Fanuc TP program (LS listing): stripped_lines.ls

/PROG  STRIPPED_TEST
/ATTR
OWNER		= MNEDITOR;
COMMENT		= "";
PROG_SIZE	= 548;
CREATE		= DATE 24-01-23  TIME 05:57:44;
MODIFIED	= DATE 25-09-11  TIME 00:54:24;
FILE_NAME	= ;
VERSION		= 0;
LINE_COUNT	= 5;
MEMORY_SIZE	= 940;
PROTECT		= READ_WRITE;
TCD:  STACK_SIZE	= 0,
      TASK_PRIORITY	= 50,
      TIME_SLICE	= 0,
      BUSY_LAMP_OFF	= 0,
      ABORT_REQUEST	= 0,
      PAUSE_REQUEST	= 0;
DEFAULT_GROUP	= 1,*,*,*,*;
CONTROL_CODE	= 00000000 00000000;
/APPL
/MN
   :  R[1]=5 ;
   :  CALL MYPROG ;
   :   ;
/POS
/END
